//{attribute 'qualified_only'}
VAR_GLOBAL CONSTANT
	//localPrgName : STRING := TO_STRING(AreaNum.AREA_4);
	//localAmsNetId : T_AmsNetId := '192.168.101.188.1.1';
	//localAmsPort : T_AmsPort := 851;
END_VAR

(* stored: Version 1.1.0.1, ProductVersion 3.1.4024.11
   GVL LocalSocket: Id {6a887490-4345-4dc6-94a1-644232984bfb} *)
